PROGRAM MAIN
VAR
END_VAR

END_PROGRAM

(* stored: Version 1.1.0.1
   POU MAIN: Id {a3d44890-e4e3-4a5f-a923-c2933341ade0} *)
